// TwinCAT 3 PLC project Tc3_MiniFrame
// Title: Tc3_MiniFrame
// Company: Gayfiles
// Author: Meisterzunge
// ProjectVersion: 0.0.0.1
// ProgramVersion: 3.1.4026.9
// libraries:
//   Tc2_Standard, * (Beckhoff Automation GmbH)
//   Tc2_System, * (Beckhoff Automation GmbH)
// project tree:
//   Events/ E_Mfr_NotifySeverity.TcDUT, FB_Mfr_Event.TcPOU (not stored), FB_Mfr_Notification.TcPOU (not stored)
//   / FB_Mfr.TcPOU (not stored)
//   Global/ Mfr_Global.TcGVL (not stored), Mfr_Param.TcGVL
//   Objects/ FB_Mfr_AI.TcPOU (not stored), FB_Mfr_AO.TcPOU (not stored), FB_Mfr_AVal.TcPOU (not stored), FB_Mfr_AValOp.TcPOU (not stored), FB_Mfr_BValOp.TcPOU (not stored), FB_Mfr_BVal.TcPOU (not stored), FB_Mfr_BI.TcPOU (not stored), FB_Mfr_BO.TcPOU (not stored), FB_Mfr_View.TcPOU, FB_Mfr_MValOp.TcPOU (not stored), FB_Mfr_MVal.TcPOU (not stored)
//   Services/Weather/ E_Mfr_WndBrng.TcDUT (not stored), E_Mfr_WthCond.TcDUT (not stored), FB_Mfr_WeatherNow.TcPOU (not stored), FB_Mfr_Weather.TcPOU (not stored), FB_Mfr_WeatherForecast.TcPOU (not stored), F_BA_IsRaining.TcPOU (not stored), I_Mfr_WeatherForecast.TcPOU, I_Mfr_WeatherNow.TcPOU
//   Universal/ E_Mfr_MeasuringElement.TcDUT (not stored)

// ---- Events/E_Mfr_NotifySeverity.TcDUT
TYPE E_Mfr_NotifySeverity :
(
	eInfo		:= 0,
	eWarning	:= 1,
	eError		:= 2
);
END_TYPE

// ---- Global/Mfr_Param.TcGVL
{attribute 'qualified_only'}
VAR_GLOBAL CONSTANT
	DefaultSensorElement : E_Mfr_MeasuringElement := E_Mfr_MeasuringElement.eNI1000;
END_VAR

// ---- Services/Weather/I_Mfr_WeatherForecast.TcPOU
/// Read-only interface exposing all output variables of FB_Mfr_WeatherForecast (including base class fields).
INTERFACE I_Mfr_WeatherForecast

/// TRUE = daytime slot, FALSE = night slot.
PROPERTY IsDaytime : BOOL
GET
END_GET
END_PROPERTY

/// Precipitation [mm].
PROPERTY Precipitation : REAL
GET
END_GET
END_PROPERTY

/// Precipitation probability [%].
PROPERTY PrecipitationProbability : REAL
GET
END_GET
END_PROPERTY

/// Temperature [°C].
PROPERTY Temperature : REAL
GET
END_GET
END_PROPERTY

/// Period low temperature [°C].
PROPERTY TemperatureLow : REAL
GET
END_GET
END_PROPERTY

/// TRUE when the gateway has written valid weather data.
PROPERTY Valid : BOOL
GET
END_GET
END_PROPERTY

/// Weather condition code.
PROPERTY WeatherCondition : E_Mfr_WthCond
GET
END_GET
END_PROPERTY

/// Wind bearing (16 cardinal directions).
PROPERTY WindBearing : E_Mfr_WndBrng
GET
END_GET
END_PROPERTY

/// Wind speed [km/h].
PROPERTY WindSpeed : REAL
GET
END_GET
END_PROPERTY

END_INTERFACE

// ---- Services/Weather/I_Mfr_WeatherNow.TcPOU
/// Read-only interface exposing all output variables of FB_Mfr_WeatherNow (including base class fields).
INTERFACE I_Mfr_WeatherNow

/// Cloud coverage [%].
PROPERTY CloudCoverage : REAL
GET
END_GET
END_PROPERTY

/// Relative humidity [%].
PROPERTY Humidity : REAL
GET
END_GET
END_PROPERTY

/// Precipitation [mm].
PROPERTY Precipitation : REAL
GET
END_GET
END_PROPERTY

/// Atmospheric pressure [hPa].
PROPERTY Pressure : REAL
GET
END_GET
END_PROPERTY

/// Temperature [°C].
PROPERTY Temperature : REAL
GET
END_GET
END_PROPERTY

/// TRUE when the gateway has written valid weather data.
PROPERTY Valid : BOOL
GET
END_GET
END_PROPERTY

/// Visibility [km].
PROPERTY Visibility : REAL
GET
END_GET
END_PROPERTY

/// Weather condition code.
PROPERTY WeatherCondition : E_Mfr_WthCond
GET
END_GET
END_PROPERTY

/// Wind bearing (16 cardinal directions).
PROPERTY WindBearing : E_Mfr_WndBrng
GET
END_GET
END_PROPERTY

/// Wind speed [km/h].
PROPERTY WindSpeed : REAL
GET
END_GET
END_PROPERTY

END_INTERFACE

// ---- Objects/FB_Mfr_View.TcPOU
// Structured view.
FUNCTION_BLOCK FB_Mfr_View EXTENDS FB_Mfr

SUPER^();

END_FUNCTION_BLOCK
